FUNCTION_BLOCK ILOCK_FB_RS (* Realizes a bistable reset-dominat latch *)
  (* Standard: 61499-1; Description: Copyright (c) 2023 Martin Erich Jobst This program and the accompanying materials are made available under the terms of the Eclipse Public License 2.0 which is available at https://www.eclipse.org/legal/epl-2.0/ SPDX-License-Identifier: EPL-2.0 *)
  (* Version 3.0, 2025-04-14, Patrick Aigner, changed package *)
  (* Version 1.0, 2023-04-28, Martin Jobst *)
  PACKAGE logiBUS::signalprocessing::interlock;
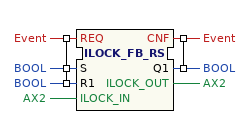
  EVENT_INPUT
    REQ WITH S, R1; (* Normal Execution Request *)
  END_EVENT
  EVENT_OUTPUT
    CNF WITH Q1; (* Execution Confirmation *)
  END_EVENT
  VAR_INPUT
    S : BOOL; (* Set *)
    R1 : BOOL; (* Reset *)
  END_VAR
  VAR_OUTPUT
    Q1 : BOOL; (* Output *)
  END_VAR
  SOCKETS
    ILOCK_IN : adapter::types::bidirectional::AX2;
  END_SOCKETS
  PLUGS
    ILOCK_OUT : adapter::types::bidirectional::AX2;
  END_PLUGS
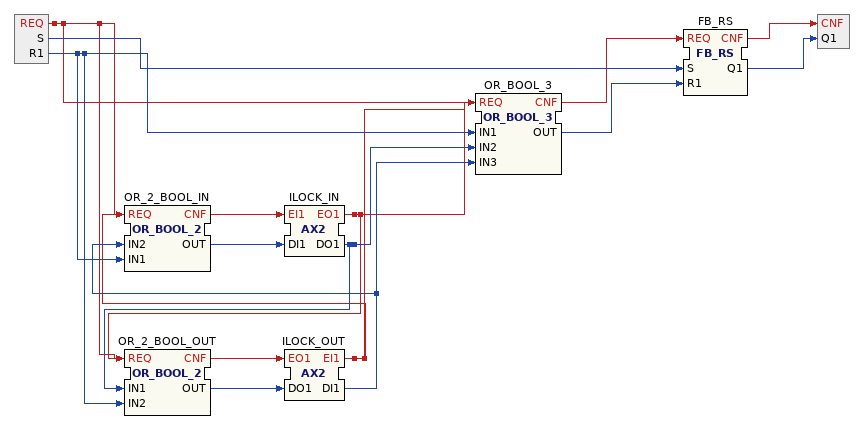
  FBS
    FB_RS : iec61131::bistableElements::FB_RS;
    OR_2_BOOL_OUT : iec61131::booleanOperators::OR_BOOL_2;
    OR_2_BOOL_IN : iec61131::booleanOperators::OR_BOOL_2;
    OR_BOOL_3 : iec61131::booleanOperators::OR_BOOL_3;
  END_FBS
  EVENT_CONNECTIONS
    REQ TO OR_BOOL_3.REQ;
    FB_RS.CNF TO CNF;
    ILOCK_OUT.EI1 TO OR_2_BOOL_IN.REQ;
    OR_2_BOOL_IN.CNF TO ILOCK_IN.EI1;
    OR_2_BOOL_OUT.CNF TO ILOCK_OUT.EO1;
    ILOCK_IN.EO1 TO OR_2_BOOL_OUT.REQ;
    REQ TO OR_2_BOOL_OUT.REQ;
    REQ TO OR_2_BOOL_IN.REQ;
    OR_BOOL_3.CNF TO FB_RS.REQ;
    ILOCK_IN.EO1 TO OR_BOOL_3.REQ;
    ILOCK_OUT.EI1 TO OR_BOOL_3.REQ;
  END_CONNECTIONS
  DATA_CONNECTIONS
    S TO FB_RS.S;
    R1 TO OR_BOOL_3.IN1;
    FB_RS.Q1 TO Q1;
    ILOCK_IN.DO1 TO OR_2_BOOL_OUT.IN1;
    OR_2_BOOL_OUT.OUT TO ILOCK_OUT.DO1;
    ILOCK_OUT.DI1 TO OR_2_BOOL_IN.IN2;
    OR_2_BOOL_IN.OUT TO ILOCK_IN.DI1;
    R1 TO OR_2_BOOL_IN.IN1;
    R1 TO OR_2_BOOL_OUT.IN2;
    OR_BOOL_3.OUT TO FB_RS.R1;
    ILOCK_IN.DO1 TO OR_BOOL_3.IN2;
    ILOCK_OUT.DI1 TO OR_BOOL_3.IN3;
  END_CONNECTIONS
END_FUNCTION_BLOCK
